PROGRAM Shutdown
VAR
	bStart	AT%I* : BOOL := FALSE;
	Shutdown_Block: NT_Shutdown;
END_VAR

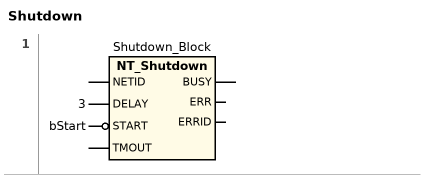
// NETWORK 1
Shutdown_Block(DELAY := 3, START := NOT bStart); // NT_Shutdown

END_PROGRAM

(* stored: Version 1.1.0.1, ProductVersion 3.1.4022.3
   POU Shutdown: Id {60141087-efde-4e46-89e7-fe8a9805e4ff}, SpecialFunc None *)
